VAR_GLOBAL
	{attribute 'TcContextId':='0'}
	fbMachine : FB_Machine; // Process cell
END_VAR

(* stored: Version 1.1.0.1, ProductVersion 3.1.4024.13
   GVL GVL_Components: Id {a65a6109-e8ab-4760-bc8a-9f6c5ab8d822} *)
